{attribute 'qualified_only'}
VAR_GLOBAL
	
	bInAckSignal	AT %I* : BOOL;

END_VAR

(* stored: Version 1.1.0.1, ProductVersion 3.1.4024.12
   GVL IO: Id {8deca2e5-e9e6-4181-a0ea-ffdba1e92be9} *)
